FUNCTION_BLOCK FB_ValveStatus
VAR_INPUT
	Input																: BOOL;
	Open																: BOOL;
	Closed																: BOOL;
	Delay																: REAL;
END_VAR
VAR_OUTPUT
	Status																: INT;
END_VAR
VAR
	Timer																: TON;
	LastInput															: BOOL;
END_VAR

// FB_ValveStatus
// Rev 1.0 - October 22, 2024

IF Input <> LastInput THEN
	LastInput															:= Input;
	Timer(IN:= FALSE);
END_IF
IF (Input AND NOT Open) OR (NOT Input AND NOT Closed) THEN
	Timer(IN:= TRUE, PT:= REAL_TO_TIME(Delay));
	IF Timer.Q THEN
		Status															:= 2;
	ELSE
		Status															:= 1;
	END_IF
ELSE
	Status																:= 0;
END_IF

END_FUNCTION_BLOCK

(* stored: Version 1.1.0.1, ProductVersion 3.1.4024.13
   POU FB_ValveStatus: Id {76d79f8f-73a0-45fe-9bcd-f6c727219450}, SpecialFunc None *)
